FUNCTION_BLOCK FB_Observable_LREAL EXTENDS FB_AbstractObservable
VAR
    _fVal:                  LREAL;
    _fOldVal:               LREAL;
END_VAR

METHOD FB_init : BOOL
VAR_INPUT
    bInitRetains:       BOOL; // if TRUE, the retain variables are initialized (warm start / cold start)
    bInCopyCode:        BOOL;  // if TRUE, the instance afterwards gets moved into the copy code (online change)
    bAutoNotify:        BOOL;
END_VAR
THIS^._nTypeClass := __SYSTEM.TYPE_CLASS.TYPE_LREAL;
END_METHOD

PROPERTY fValue64 : LREAL
GET
fValue64 := THIS^._fVal;
END_GET
SET
THIS^._fOldVal := _fVal;
THIS^._fVal := fValue64;

THIS^.NotifyWithConditions();
END_SET
END_PROPERTY

PROPERTY nDataSize : UDINT
GET
nDataSize := SIZEOF(LREAL);
END_GET
END_PROPERTY

PROPERTY PROTECTED pData : POINTER TO BYTE
GET
pData := ADR(THIS^._fVal);
END_GET
END_PROPERTY

METHOD  ValueChanged : BOOL
VAR_INPUT
END_VAR
ValueChanged := THIS^._fOldVal <> THIS^._fVal;
END_METHOD

END_FUNCTION_BLOCK

(* stored: Version 1.1.0.1, ProductVersion 3.1.4024.12
   POU FB_Observable_LREAL: Id {fa67ef6a-ec89-437e-b171-e4161c6cb780}, SpecialFunc None
   Method FB_init: Id {f5811821-f706-0836-1f4d-4ec5226e116e}
   Property fValue64: Id {69f3a879-ee85-4896-b924-fb4f518a4add}
   Get Get: Id {3f8ddbf1-df60-462a-9afe-0be07f6ff38b}
   Set Set: Id {f4f1b1f9-183d-4a8e-852f-d366e51e67ca}
   Property nDataSize: Id {4a01f3e2-fc6a-4cac-b7bf-b51b8920eff6}
   Get Get: Id {abfd40cb-2260-4d70-8767-dd05299575a7}
   Property pData: Id {7840c422-cf8a-4191-9426-4f5ea5c99cfb}
   Get Get: Id {522cfd57-e430-438a-b54c-ae6d1ebe9b9b}
   Method ValueChanged: Id {4bb64c16-6708-008b-1182-b25cbfc886cd} *)
